FUNCTION_BLOCK FB_Professor

VAR
	
    sName   : STRING := '';
    sOutput : STRING := '';
END_VAR

METHOD GetName :  STRING
VAR_INPUT
END_VAR
GetName := sName;
END_METHOD

METHOD SetName 
VAR_INPUT
	    sInputName : STRING;

END_VAR
sName := sInputName;
END_METHOD

END_FUNCTION_BLOCK

(* stored: Version 1.1.0.1, ProductVersion 3.1.4024.16
   POU FB_Professor: Id {00c1dd9b-40c8-4f24-a3e5-cfecc2666d09}, SpecialFunc None
   Method GetName: Id {f70eb46d-ad49-4a39-a018-5f95f50b4a46}
   Method SetName: Id {2cd17729-460f-4124-a775-4f07df511011} *)
